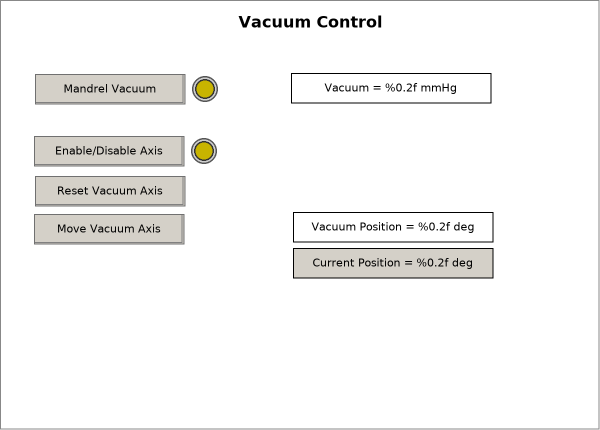
VISUALIZATION Manual_Vacuum  // 600x430
    Label (133,7 355x30), "Vacuum Control"
    Rectangle (291,73 200x30), "Vacuum = %0.2f mmHg", text variable: MAIN.fbSlitter.Mandrel._vacuum_mmHg
    Button (35,74 150x30), "Mandrel Vacuum"
        OnMouseClick: execute { MAIN.fbSlitter.Manual.bToggleMandrelVacuum := TRUE; }
    Lamp1 (190,74 30x30), variable: MAIN.fbSlitter.Mandrel.doVacuum, style: Lamp-Lamp1-Yellow
    Button (34,136 150x30), "Enable/Disable Axis"
        OnMouseClick: execute { MAIN.fbSlitter.Manual.bVacuumAxisToggleEnable := TRUE; }
    Lamp1 (189,136 30x30), variable: MAIN.fbSlitter.Mandrel.VacAxis.axis.NcToPlc.StateDWord.0 = 1, style: Lamp-Lamp1-Yellow
    Rectangle (293,248 200x30), "Current Position = %0.2f deg", text variable: MAIN.fbSlitter.Mandrel.VacAxis.axis.NcToPlc.ActPos
    Rectangle (293,212 200x30), "Vacuum Position = %0.2f deg", text variable: MAIN.TubeHmi.VacPosition
        OnMouseClick: write MAIN.TubeHmi.VacPosition via Default, min 0, max 13000, title 'Vacuum Position'
    Button (34,214 150x30), "Move Vacuum Axis"
        OnMouseClick: execute { MAIN.fbSlitter.Manual.bVacuumAxisMove := TRUE; }
    Button (35,176 150x30), "Reset Vacuum Axis"
        OnMouseClick: execute { MAIN.fbSlitter.Manual.bVacuumAxisReset := TRUE; }
END_VISUALIZATION

(* stored: Version 1.1.0.1, ProductVersion 3.1.4024.9
   Visu Manual_Vacuum: Id {ec2aa9d7-6a57-4309-90ec-3835c2701fc4} *)
